(* IEC 61131-3 sources: JaccoSigma/tempclass/Class/DSComm_Interface (part 2) *)

#pragma usingLtd DSComm

#pragma using DSComm

FUNCTION GLOBAL DSComm_Interface::GetVersion
	VAR_OUTPUT
		MessageID 	: DINT;
	END_VAR

  MessageID := DSComm.GetVersion(pThis:=this);
END_FUNCTION

#pragma warning(disable: 73)
FUNCTION VIRTUAL GLOBAL DSComm_Interface::GetVersionResp
	VAR_INPUT
		MessageID 	: DINT;
		ErrorNo 	: DINT;
		pGetVersionRsp 	: ^DSComm::_DS_GetVersionResp;
	END_VAR
#pragma warning(default: 73)

END_FUNCTION

#pragma warning(disable: 73)

#pragma warning(disable: 73)
FUNCTION VIRTUAL GLOBAL DSComm_Interface::GetProjectInfoResp
	VAR_INPUT
		MessageID 	: DINT;
		ErrorNo 	: DINT;
		pGetProjectInfoRsp 	: ^DSComm::_DS_GetProjectInfoResp;
	END_VAR
#pragma warning(default: 73)

END_FUNCTION

FUNCTION GLOBAL DSComm_Interface::UserLogin
	VAR_INPUT
		pUserName 	: ^UINT;
		pPassword 	: ^UINT;
	END_VAR
	VAR_OUTPUT
		MessageID 	: DINT;
	END_VAR

  MessageID := DSComm.UserLogin(pThis:=this, pUserName, pPassword);
END_FUNCTION

#pragma warning(disable: 73)
FUNCTION VIRTUAL GLOBAL DSComm_Interface::UserLoginResp
	VAR_INPUT
    MessageID   : DINT;
    ErrorNo     : DINT;
    pUserLoginData : ^DSComm::_DS_UserLoginResp;
	END_VAR
#pragma warning(default: 73)

END_FUNCTION

FUNCTION GLOBAL DSComm_Interface::GetValue
	VAR_INPUT
		num 	: UDINT;
		pGetValue 	: ^DSComm::_DS_GetValueCmd;
	END_VAR
	VAR_OUTPUT
		MessageID 	: DINT;
	END_VAR

  MessageID := DSComm.GetValue(pThis:=this, num, pGetValue);
END_FUNCTION

#pragma warning(disable: 73)
FUNCTION VIRTUAL GLOBAL DSComm_Interface::GetValueResp
VAR_INPUT
    MessageID   : DINT;
    ErrorNo     : DINT;
    num         : UDINT;
    pGetValueRsp: ^DSComm::_DS_GetValueResp;
END_VAR
#pragma warning(default: 73)

END_FUNCTION

FUNCTION GLOBAL DSComm_Interface::SetValue
	VAR_INPUT
		num 	: UDINT;
		pSetValue 	: ^DSComm::_DS_SetValueCmd;
	END_VAR
	VAR_OUTPUT
		MessageID 	: DINT;
	END_VAR

  MessageID := DSComm.SetValue(pThis:=this, num, pSetValue);
END_FUNCTION

#pragma warning(disable: 73)
FUNCTION VIRTUAL GLOBAL DSComm_Interface::SetValueResp
VAR_INPUT
    MessageID   : DINT;
    ErrorNo     : DINT;
    num         : UDINT;
    pSetValueRsp: ^DSComm::_DS_SetValueResp;
END_VAR
#pragma warning(default: 73)

END_FUNCTION

FUNCTION GLOBAL DSComm_Interface::GetString
	VAR_INPUT
		num 	: UDINT;
		pGetString 	: ^DSComm::_DS_GetStringCmd;
	END_VAR
	VAR_OUTPUT
		MessageID 	: DINT;
	END_VAR

  MessageID := DSComm.GetString(pThis:=this, num, pGetString);
END_FUNCTION

#pragma warning(disable: 73)
FUNCTION VIRTUAL GLOBAL DSComm_Interface::GetStringResp
VAR_INPUT
    MessageID   : DINT;
    ErrorNo     : DINT;
    num         : UDINT;
    pGetStringRsp: ^DSComm::_DS_GetStringResp;
END_VAR
#pragma warning(default: 73)

END_FUNCTION

FUNCTION GLOBAL DSComm_Interface::SetString
	VAR_INPUT
		num 	: UDINT;
		pSetString 	: ^DSComm::_DS_SetStringCmd;
	END_VAR
	VAR_OUTPUT
		MessageID 	: DINT;
	END_VAR

  MessageID := DSComm.SetString(pThis:=this, num, pSetString);
END_FUNCTION

#pragma warning(disable: 73)
FUNCTION VIRTUAL GLOBAL DSComm_Interface::SetStringResp
VAR_INPUT
    MessageID   : DINT;
    ErrorNo     : DINT;
    num         : UDINT;
    pSetStringRsp: ^DSComm::_DS_SetStringResp;
END_VAR
#pragma warning(default: 73)

END_FUNCTION

FUNCTION GLOBAL DSComm_Interface::CancelCommand
	VAR_INPUT
		HandleID 	: DINT;
	END_VAR
	VAR_OUTPUT
		MessageID 	: DINT;
	END_VAR

  MessageID := DSComm.CancelCommand(pThis:=this, HandleID$UDINT);
  MessageID += 1;
END_FUNCTION

#pragma warning(disable: 73)
FUNCTION VIRTUAL GLOBAL DSComm_Interface::CancelCommandResp
	VAR_INPUT
		MessageID 	: DINT;
		ErrorNo 	: DINT;
		pCancelRsp 	: ^DSComm::_DS_CancelResp;
	END_VAR
#pragma warning(default: 73)

END_FUNCTION

FUNCTION GLOBAL DSComm_Interface::Loop
	VAR_INPUT
		Station 	: UDINT;
		pDataSrc 	: pVoid;
		DataLen 	: UDINT;
	END_VAR
	VAR_OUTPUT
		MessageID 	: DINT;
	END_VAR

  MessageID := DSComm.Loop(pThis:=this, Station, pDataSrc, DataLen);
END_FUNCTION

#pragma warning(disable: 73)
FUNCTION VIRTUAL GLOBAL DSComm_Interface::LoopResp
	VAR_INPUT
		MessageID 	: DINT;
		ErrorNo 	: DINT;
		Station 	: UDINT;
		pData 	: pVoid;
		Length 	: UDINT;
	END_VAR
#pragma warning(default: 73)

END_FUNCTION

FUNCTION GLOBAL DSComm_Interface::RecipeLoad
	VAR_INPUT
		pFilterIncl 	: ^DSComm::_DS_UnsLongLongInt;
		pFilterExcl 	: ^DSComm::_DS_UnsLongLongInt;
		crc 	: UDINT;
		pDpne 	: ^CHAR;
	END_VAR
	VAR_OUTPUT
		MessageID 	: DINT;
	END_VAR

  MessageID := DSComm.RecipeLoad(pThis:=this, pFilterIncl, pFilterExcl, crc, pDpne);
END_FUNCTION

#pragma warning(disable: 73)
FUNCTION VIRTUAL GLOBAL DSComm_Interface::RecipeLoadResp
	VAR_INPUT
		MessageID 	: DINT;
		ErrorNo 	: DINT;
		pRecipeLoadRsp 	: ^DSComm::_DS_RecipeLoadResp;
	END_VAR
#pragma warning(default: 73)

END_FUNCTION

FUNCTION GLOBAL DSComm_Interface::RecipeSave
	VAR_INPUT
		pFilterIncl 	: ^DSComm::_DS_UnsLongLongInt;
		pFilterExcl 	: ^DSComm::_DS_UnsLongLongInt;
		pDpne 	: ^CHAR;
		pHeaderText 	: ^CHAR;
	END_VAR
	VAR_OUTPUT
		MessageID 	: DINT;
	END_VAR

  MessageID := DSComm.RecipeSave(pThis:=this, pFilterIncl, pFilterExcl, pDpne, pHeaderText);
END_FUNCTION

#pragma warning(disable: 73)
FUNCTION VIRTUAL GLOBAL DSComm_Interface::RecipeSaveResp
	VAR_INPUT
		MessageID 	: DINT;
		ErrorNo 	: DINT;
		pRecipeSaveRsp 	: ^DSComm::_DS_RecipeSaveResp;
	END_VAR
#pragma warning(default: 73)

END_FUNCTION

FUNCTION GLOBAL DSComm_Interface::SendToAll
	VAR_INPUT
		pDataSrc 	: pVoid;
		DataLen 	: UDINT;
	END_VAR
	VAR_OUTPUT
		MessageID 	: DINT;
	END_VAR

  MessageID := DSComm.SendToAll(pThis:=this, pDataSrc, DataLen);
END_FUNCTION

#pragma warning(disable: 73)
FUNCTION VIRTUAL GLOBAL DSComm_Interface::SendToAllResp
VAR_INPUT
    MessageID   : DINT;
    ErrorNo     : DINT;
END_VAR
#pragma warning(default: 73)

END_FUNCTION

FUNCTION GLOBAL DSComm_Interface::UserLogout
	VAR_OUTPUT
		MessageID 	: DINT;
	END_VAR

  MessageID := DSComm.UserLogout(pThis:=this);
END_FUNCTION

#pragma warning(disable: 73)
FUNCTION VIRTUAL GLOBAL DSComm_Interface::UserLogoutResp
VAR_INPUT
    MessageID   : DINT;
    ErrorNo     : DINT;
END_VAR
#pragma warning(default: 73)

END_FUNCTION

FUNCTION GLOBAL DSComm_Interface::UserPasswordChange
	VAR_INPUT
		pOldPassword 	: ^UINT;
		pNewPassword 	: ^UINT;
	END_VAR
	VAR_OUTPUT
		MessageID 	: DINT;
	END_VAR

  MessageID := DSComm.UserPasswordChange(pThis:=this, pOldPassword, pNewPassword);
END_FUNCTION

#pragma warning(disable: 73)
FUNCTION VIRTUAL GLOBAL DSComm_Interface::UserPasswordChangeResp
	VAR_INPUT
		MessageID 	: DINT;
		ErrorNo 	: DINT;
		pUserPasswordChangeRsp 	: ^DSComm::_DS_UserPasswordChangeResp;
	END_VAR
#pragma warning(default: 73)

END_FUNCTION

FUNCTION GLOBAL DSComm_Interface::CheckAccessLevel
	VAR_INPUT
		num 	: UDINT;
		pCheckAccessLevel 	: ^DSComm::_DS_CheckAccessLevelCmd;
	END_VAR
	VAR_OUTPUT
		MessageID 	: DINT;
	END_VAR

  MessageID := DSComm.CheckAccessLevel(pThis:=this, num, pCheckAccessLevel);
END_FUNCTION

#pragma warning(disable: 73)
FUNCTION VIRTUAL GLOBAL DSComm_Interface::CheckAccessLevelResp
	VAR_INPUT
		MessageID 	: DINT;
		ErrorNo 	: DINT;
		num 	: UDINT;
		pCheckAccessLevelRsp 	: ^DSComm::_DS_CheckAccessLevelResp;
	END_VAR
#pragma warning(default: 73)

END_FUNCTION

FUNCTION GLOBAL DSComm_Interface::CreateUser
	VAR_INPUT
		num 	: UDINT;
		pCreateUser 	: ^DSComm::_DS_CreateUserCmd;
	END_VAR
	VAR_OUTPUT
		MessageID 	: DINT;
	END_VAR

  MessageID := DSComm.CreateUser(pThis:=this, num, pCreateUser);
END_FUNCTION

#pragma warning(disable: 73)
FUNCTION VIRTUAL GLOBAL DSComm_Interface::CreateUserResp
VAR_INPUT
    MessageID   : DINT;
    ErrorNo     : DINT;
    num         : UDINT;
    pCreateUserRsp : ^DSComm::_DS_CreateUserResp;
END_VAR
#pragma warning(default: 73)

END_FUNCTION

FUNCTION GLOBAL DSComm_Interface::ChangeUserSettings
	VAR_INPUT
		num 	: UDINT;
		pChangeUsrSettings 	: ^DSComm::_DS_ChangeUserSettingsCmd;
	END_VAR
	VAR_OUTPUT
		MessageID 	: DINT;
	END_VAR

  MessageID := DSComm.ChangeUserSettings(pThis:=this, num, pChangeUsrSettings);
END_FUNCTION

#pragma warning(disable: 73)
FUNCTION VIRTUAL GLOBAL DSComm_Interface::ChangeUserSettingsResp
	VAR_INPUT
		MessageID 	: DINT;
		ErrorNo 	: DINT;
		num 	: UDINT;
		pChangeUserRsp 	: ^DSComm::_DS_ChangeUserSettingsResp;
	END_VAR
#pragma warning(default: 73)

END_FUNCTION

FUNCTION GLOBAL DSComm_Interface::DeleteUser
	VAR_INPUT
		num 	: UDINT;
		pUserID 	: ^UDINT;
	END_VAR
	VAR_OUTPUT
		MessageID 	: DINT;
	END_VAR

  MessageID := DSComm.DeleteUser(pThis:=this, num, pUserID);
END_FUNCTION

#pragma warning(disable: 73)
FUNCTION VIRTUAL GLOBAL DSComm_Interface::DeleteUserResp
VAR_INPUT
    MessageID   : DINT;
    ErrorNo     : DINT;
    num         : UDINT;
    pDeleteUserRsp : ^DSComm::_DS_DeleteUserResp;
END_VAR
#pragma warning(default: 73)

END_FUNCTION

FUNCTION GLOBAL DSComm_Interface::GetUserList
	VAR_OUTPUT
		MessageID 	: DINT;
	END_VAR

  MessageID := DSComm.GetUserList(pThis:=this);
END_FUNCTION

#pragma warning(disable: 73)
FUNCTION VIRTUAL GLOBAL DSComm_Interface::GetUserListResp
VAR_INPUT
    MessageID   : DINT;
    ErrorNo     : DINT;
    num         : UDINT;
    pGetUserListRsp: ^DSComm::_DS_GetUserListResp;
END_VAR
#pragma warning(default: 73)

END_FUNCTION

FUNCTION GLOBAL DSComm_Interface::GetUserDetails
	VAR_INPUT
		userID 	: UDINT;
	END_VAR
	VAR_OUTPUT
		MessageID 	: DINT;
	END_VAR

  MessageID := DSComm.GetUserDetails(pThis:=this, userID);
END_FUNCTION

#pragma warning(disable: 73)
FUNCTION VIRTUAL GLOBAL DSComm_Interface::GetUserDetailsResp
	VAR_INPUT
		MessageID 	: DINT;
		ErrorNo 	: DINT;
		pUserDetails 	: ^DSComm::_DS_UserLoginResp;
	END_VAR
#pragma warning(default: 73)

END_FUNCTION

FUNCTION GLOBAL DSComm_Interface::CreateRole
	VAR_INPUT
		num 	: UDINT;
		pCreateRolePara 	: ^DSComm::_DS_CreateRoleCmd;
	END_VAR
	VAR_OUTPUT
		MessageID 	: DINT;
	END_VAR

  MessageID := DSComm.CreateRole(pThis:=this, num, pCreateRolePara);
END_FUNCTION

#pragma warning(disable: 73)
FUNCTION VIRTUAL GLOBAL DSComm_Interface::CreateRoleResp
VAR_INPUT
    MessageID   : DINT;
    ErrorNo     : DINT;
    num         : UDINT;
    pCreateRoleRsp : ^DSComm::_DS_CreateRoleResp;
END_VAR
#pragma warning(default: 73)

END_FUNCTION

FUNCTION GLOBAL DSComm_Interface::ChangeRole
	VAR_INPUT
		num 	: UDINT;
		pChangeRole 	: ^DSComm::_DS_ChangeRoleCmd;
	END_VAR
	VAR_OUTPUT
		MessageID 	: DINT;
	END_VAR

  MessageID := DSComm.ChangeRole(pThis:=this, num, pChangeRole);
END_FUNCTION

#pragma warning(disable: 73)
FUNCTION VIRTUAL GLOBAL DSComm_Interface::ChangeRoleResp
VAR_INPUT
    MessageID   : DINT;
    ErrorNo     : DINT;
    num         : UDINT;
    pChangeRoleRsp : ^DSComm::_DS_ChangeRoleResp;
END_VAR
#pragma warning(default: 73)

END_FUNCTION

FUNCTION GLOBAL DSComm_Interface::DeleteRole
	VAR_INPUT
		num 	: UDINT;
		pRoleID 	: ^UDINT;
	END_VAR
	VAR_OUTPUT
		MessageID 	: DINT;
	END_VAR

  MessageID := DSComm.DeleteRole(pThis:=this, num, pRoleID);
END_FUNCTION

#pragma warning(disable: 73)
FUNCTION VIRTUAL GLOBAL DSComm_Interface::DeleteRoleResp
VAR_INPUT
    MessageID   : DINT;
    ErrorNo     : DINT;
    num         : UDINT;
    pDeleteRoleRsp : ^DSComm::_DS_DeleteRoleResp;
END_VAR
#pragma warning(default: 73)

END_FUNCTION

FUNCTION GLOBAL DSComm_Interface::GetRoleList
	VAR_OUTPUT
		MessageID 	: DINT;
	END_VAR

  MessageID := DSComm.GetRoleList(pThis:=this);
END_FUNCTION

#pragma warning(disable: 73)
FUNCTION VIRTUAL GLOBAL DSComm_Interface::GetRoleListResp
VAR_INPUT
    MessageID   : DINT;
    ErrorNo     : DINT;
    num         : UDINT;
    pGetRoleListRsp: ^DSComm::_DS_GetRoleListResp;
END_VAR
#pragma warning(default: 73)

END_FUNCTION

FUNCTION GLOBAL DSComm_Interface::GetRoleDetails
	VAR_INPUT
		roleID 	: UDINT;
	END_VAR
	VAR_OUTPUT
		MessageID 	: DINT;
	END_VAR

  MessageID := DSComm.GetRoleDetails(pThis:=this, roleID);
END_FUNCTION

#pragma warning(disable: 73)
FUNCTION VIRTUAL GLOBAL DSComm_Interface::GetRoleDetailsResp
VAR_INPUT
    MessageID   : DINT;
    ErrorNo     : DINT;
    pGetRoleDetailsRsp : ^DSComm::_DS_GetRoleDetailsResp;
END_VAR
#pragma warning(default: 73)

END_FUNCTION

FUNCTION GLOBAL DSComm_Interface::GetVarIdFromName
	VAR_INPUT
		num 	: UDINT;
		ppName 	: ^pChar;
	END_VAR
	VAR_OUTPUT
		MessageID 	: DINT;
	END_VAR

  MessageID := DSComm.GetVarIdFromName(pThis:=this, num, ppName);
END_FUNCTION

#pragma warning(disable: 73)
FUNCTION VIRTUAL GLOBAL DSComm_Interface::GetVarIdFromNameResp
VAR_INPUT
    MessageID   : DINT;
    ErrorNo     : DINT;
    num         : UDINT;
    pGetVarIdFromNameRsp: ^DSComm::_DS_GetVarIdFromNameResp;
END_VAR
#pragma warning(default: 73)

END_FUNCTION

FUNCTION GLOBAL DSComm_Interface::GetVarIdFromLasalId
	VAR_INPUT
		num 	: UDINT;
		pLasalId 	: ^DSComm::_DS_GetVarIdFromLasalIdCmd;
	END_VAR
	VAR_OUTPUT
		MessageID 	: DINT;
	END_VAR

  MessageID := DSComm.GetVarIdFromLasalId(pThis:=this, num, pLasalId);
END_FUNCTION

#pragma warning(disable: 73)
FUNCTION VIRTUAL GLOBAL DSComm_Interface::GetVarIdFromLasalIdResp
VAR_INPUT
    MessageID   : DINT;
    ErrorNo     : DINT;
    num         : UDINT;
    pGetVarIdFromLasalIdRsp: ^DSComm::_DS_GetVarIdFromLasalIdResp;
END_VAR
#pragma warning(default: 73)

END_FUNCTION

FUNCTION GLOBAL DSComm_Interface::GetLasalIdFromName
	VAR_INPUT
		num 	: UDINT;
		ppName 	: ^pChar;
	END_VAR
	VAR_OUTPUT
		MessageID 	: DINT;
	END_VAR

  MessageID := DSComm.GetLasalIdFromName(pThis:=this, num, ppName);
END_FUNCTION

#pragma warning(disable: 73)
FUNCTION VIRTUAL GLOBAL DSComm_Interface::GetLasalIdFromNameResp
VAR_INPUT
    MessageID   : DINT;
    ErrorNo     : DINT;
    num         : UDINT;
    pGetLasalIdFromNameRsp: ^DSComm::_DS_GetLasalIdFromNameResp;
END_VAR
#pragma warning(default: 73)

END_FUNCTION

FUNCTION GLOBAL DSComm_Interface::GetLasalIdFromVarId
	VAR_INPUT
		num 	: UDINT;
		pVarId 	: ^UDINT;
	END_VAR
	VAR_OUTPUT
		MessageID 	: DINT;
	END_VAR

  MessageID := DSComm.GetLasalIdFromVarId(pThis:=this, num, pVarId);
END_FUNCTION

#pragma warning(disable: 73)
FUNCTION VIRTUAL GLOBAL DSComm_Interface::GetLasalIdFromVarIdResp
VAR_INPUT
    MessageID   : DINT;
    ErrorNo     : DINT;
    num         : UDINT;
    pGetLasalIdIdFromVarIdRsp: ^DSComm::_DS_GetLasalIdIdFromVarIdResp;
END_VAR
#pragma warning(default: 73)

END_FUNCTION

FUNCTION GLOBAL DSComm_Interface::GetNameFromVarId
	VAR_INPUT
		num 	: UDINT;
		pVarId 	: ^UDINT;
	END_VAR
	VAR_OUTPUT
		MessageID 	: DINT;
	END_VAR

  MessageID := DSComm.GetNameFromVarId(pThis:=this, num, pVarId);
END_FUNCTION

#pragma warning(disable: 73)
FUNCTION VIRTUAL GLOBAL DSComm_Interface::GetNameFromVarIdResp
VAR_INPUT
    MessageID   : DINT;
    ErrorNo     : DINT;
    num         : UDINT;
    pGetNameFromVarIdRsp: ^DSComm::_DS_GetNameFromVarIdResp;
END_VAR
#pragma warning(default: 73)

END_FUNCTION

FUNCTION GLOBAL DSComm_Interface::GetNameFromLasalId
	VAR_INPUT
		num 	: UDINT;
		pLasalId 	: ^DSComm::_DS_GetNameFromLasalIdCmd;
	END_VAR
	VAR_OUTPUT
		MessageID 	: DINT;
	END_VAR

  MessageID := DSComm.GetNameFromLasalId(pThis:=this, num, pLasalId);
END_FUNCTION

#pragma warning(disable: 73)
FUNCTION VIRTUAL GLOBAL DSComm_Interface::GetNameFromLasalIdResp
VAR_INPUT
    MessageID   : DINT;
    ErrorNo     : DINT;
    num         : UDINT;
    pGetNameFromLasalIdRsp: ^DSComm::_DS_GetNameFromLasalIdResp;
END_VAR
#pragma warning(default: 73)

END_FUNCTION

FUNCTION GLOBAL DSComm_Interface::IncValue
	VAR_INPUT
		num 	: UDINT;
		pdpId : ^UDINT;
	END_VAR
	VAR_OUTPUT
		MessageID 	: DINT;
	END_VAR

  MessageID := DSComm.IncValue(pThis:=this, num, pdpId);
END_FUNCTION

#pragma warning(disable: 73)
FUNCTION VIRTUAL GLOBAL DSComm_Interface::IncValueResp
VAR_INPUT
    MessageID   : DINT;
    ErrorNo     : DINT;
    num         : UDINT;
    pIncValueRsp: ^DSComm::_DS_IncDecValueResp;
END_VAR
#pragma warning(default: 73)

END_FUNCTION

FUNCTION GLOBAL DSComm_Interface::DecValue
	VAR_INPUT
		num 	: UDINT;
		pdpId : ^UDINT;
	END_VAR
	VAR_OUTPUT
		MessageID 	: DINT;
	END_VAR

  MessageID := DSComm.DecValue(pThis:=this, num, pdpId);
END_FUNCTION

#pragma warning(disable: 73)
FUNCTION VIRTUAL GLOBAL DSComm_Interface::DecValueResp
VAR_INPUT
    MessageID   : DINT;
    ErrorNo     : DINT;
    num         : UDINT;
    pDecValueRsp: ^DSComm::_DS_IncDecValueResp;
END_VAR
#pragma warning(default: 73)

END_FUNCTION

FUNCTION GLOBAL DSComm_Interface::RefListAdd
	VAR_INPUT
		channel 	: UDINT;
		num 	: UDINT;
		pDpId 	: ^UDINT;
	END_VAR
	VAR_OUTPUT
		MessageID 	: DINT;
	END_VAR

  MessageID := DSComm.RefListAdd(pThis:=this, channel, num, pDpId);
END_FUNCTION

#pragma warning(disable: 73)
FUNCTION VIRTUAL GLOBAL DSComm_Interface::RefListAddResp
	VAR_INPUT
		MessageID 	: DINT;
		ErrorNo 	: DINT;
		Channel 	: UDINT;
		num 	: UDINT;
		pRefListAddRsp 	: ^DSComm::_DS_RefListAddResp;
	END_VAR
#pragma warning(default: 73)

END_FUNCTION

FUNCTION GLOBAL DSComm_Interface::RefListSub
	VAR_INPUT
		channel 	: UDINT;
		num 	: UDINT;
		pDpId 	: ^UDINT;
	END_VAR
	VAR_OUTPUT
		MessageID 	: DINT;
	END_VAR

  MessageID := DSComm.RefListSub(pThis:=this, channel, num, pDpId);
END_FUNCTION

#pragma warning(disable: 73)
FUNCTION VIRTUAL GLOBAL DSComm_Interface::RefListSubResp
	VAR_INPUT
		MessageID 	: DINT;
		ErrorNo 	: DINT;
		Channel 	: UDINT;
		num 	: UDINT;
		pRefListSubRsp 	: ^DSComm::_DS_RefListSubResp;
	END_VAR
#pragma warning(default: 73)

END_FUNCTION

#pragma warning(disable: 73)
FUNCTION VIRTUAL GLOBAL DSComm_Interface::RefListUpdatePush
	VAR_INPUT
		ErrorNo 	: DINT;
		channel 	: UDINT;
		num 	: UDINT;
		pRefListUpdate 	: ^DSComm::_DS_RefListUpdate;
	END_VAR
#pragma warning(default: 73)

END_FUNCTION

#pragma warning(disable: 73)
FUNCTION VIRTUAL GLOBAL DSComm_Interface::RefListUpdateStringPush
	VAR_INPUT
		ErrorNo 	: DINT;
		channel 	: UDINT;
		num 	: UDINT;
		pRefListUpdateString 	: ^DSComm::_DS_RefListUpdateString;
	END_VAR
#pragma warning(default: 73)

END_FUNCTION

FUNCTION GLOBAL DSComm_Interface::GetDpInfo
	VAR_INPUT
		num 	: UDINT;
		pVarId 	: ^UDINT;
	END_VAR
	VAR_OUTPUT
		MessageID 	: DINT;
	END_VAR

  MessageID := DSComm.GetDpInfo(pThis:=this, num, pVarId);
END_FUNCTION

#pragma warning(disable: 73)
FUNCTION VIRTUAL GLOBAL DSComm_Interface::GetDpInfoResp
VAR_INPUT
    MessageID   : DINT;
    ErrorNo     : DINT;
    num         : UDINT;
    pGetDpInfoRsp: ^DSComm::_DS_GetDpInfoResp;
END_VAR
#pragma warning(default: 73)

END_FUNCTION

FUNCTION GLOBAL DSComm_Interface::GetDpList
	VAR_INPUT
		pFilterIncl 	: ^DSComm::_DS_UnsLongLongInt;
		pFilterExcl 	: ^DSComm::_DS_UnsLongLongInt;
	END_VAR
	VAR_OUTPUT
		MessageID 	: DINT;
	END_VAR

  MessageID := DSComm.GetDpList(pThis:=this, pFilterIncl, pFilterExcl);
END_FUNCTION

#pragma warning(disable: 73)
FUNCTION VIRTUAL GLOBAL DSComm_Interface::GetDpListResp
	VAR_INPUT
		MessageID 	: DINT;
		ErrorNo 	: DINT;
		TotalNum 	: UDINT;
		num 	: UDINT;
		LastPacket 	: BOOL;
		pGetDpListRsp 	: ^DSComm::_DS_GetDpListResp;
	END_VAR
#pragma warning(default: 73)

END_FUNCTION

#pragma warning(disable: 73)

#pragma warning(disable: 73)

FUNCTION GLOBAL DSComm_Interface::FileOpen
	VAR_INPUT
		pDpne 	: ^CHAR;
		pMode 	: ^CHAR;
	END_VAR
	VAR_OUTPUT
		MessageID 	: DINT;
	END_VAR

  MessageID := DSComm.FileOpen(pThis:=this, pDpne, pMode);
END_FUNCTION

#pragma warning(disable: 73)
FUNCTION VIRTUAL GLOBAL DSComm_Interface::FileOpenResp
VAR_INPUT
    MessageID   : DINT;
    ErrorNo     : DINT;
    pFileOpenRsp: ^DSComm::_DS_FileOpenResp;
END_VAR
#pragma warning(default: 73)

END_FUNCTION

FUNCTION GLOBAL DSComm_Interface::FileClose
	VAR_INPUT
		handle 	: UDINT;
	END_VAR
	VAR_OUTPUT
		MessageID 	: DINT;
	END_VAR

  MessageID := DSComm.FileClose(pThis:=this, handle);
END_FUNCTION

#pragma warning(disable: 73)
FUNCTION VIRTUAL GLOBAL DSComm_Interface::FileCloseResp
VAR_INPUT
    MessageID   : DINT;
    ErrorNo     : DINT;
    pFileCloseRsp: ^DSComm::_DS_FileCloseResp;
END_VAR
#pragma warning(default: 73)

END_FUNCTION

FUNCTION GLOBAL DSComm_Interface::FileSeek
	VAR_INPUT
		handle 	: UDINT;
		start 	: UDINT;
		offset 	: UDINT;
	END_VAR
	VAR_OUTPUT
		MessageID 	: DINT;
	END_VAR

  MessageID := DSComm.FileSeek(pThis:=this, handle, start, offset);
END_FUNCTION

#pragma warning(disable: 73)
FUNCTION VIRTUAL GLOBAL DSComm_Interface::FileSeekResp
VAR_INPUT
    MessageID   : DINT;
    ErrorNo     : DINT;
    pFileSeekRsp: ^DSComm::_DS_FileSeekResp;
END_VAR
#pragma warning(default: 73)

END_FUNCTION

FUNCTION GLOBAL DSComm_Interface::FileTell
	VAR_INPUT
		handle 	: UDINT;
	END_VAR
	VAR_OUTPUT
		MessageID 	: DINT;
	END_VAR

  MessageID := DSComm.FileTell(pThis:=this, handle);
END_FUNCTION

#pragma warning(disable: 73)
FUNCTION VIRTUAL GLOBAL DSComm_Interface::FileTellResp
	VAR_INPUT
		MessageID 	: DINT;
		ErrorNo 	: DINT;
		pFileTellRsp 	: ^DSComm::_DS_FileTellResp;
	END_VAR
#pragma warning(default: 73)

END_FUNCTION

FUNCTION GLOBAL DSComm_Interface::FileRead
	VAR_INPUT
		handle 	: UDINT;
		length 	: UDINT;
	END_VAR
	VAR_OUTPUT
		MessageID 	: DINT;
	END_VAR

  MessageID := DSComm.FileRead(pThis:=this, handle, length);
END_FUNCTION

#pragma warning(disable: 73)
FUNCTION VIRTUAL GLOBAL DSComm_Interface::FileReadResp
VAR_INPUT
    MessageID   : DINT;
    ErrorNo     : DINT;
    pFileReadRsp: ^DSComm::_DS_FileReadResp;
END_VAR
#pragma warning(default: 73)

END_FUNCTION

FUNCTION GLOBAL DSComm_Interface::FileWrite
	VAR_INPUT
		handle 	: UDINT;
		length 	: UDINT;
		pWriteData 	: ^CHAR;
	END_VAR
	VAR_OUTPUT
		MessageID 	: DINT;
	END_VAR

  MessageID := DSComm.FileWrite(pThis:=this, handle, length, pWriteData);
END_FUNCTION

#pragma warning(disable: 73)
FUNCTION VIRTUAL GLOBAL DSComm_Interface::FileWriteResp
VAR_INPUT
    MessageID   : DINT;
    ErrorNo     : DINT;
    pFileWriteRsp: ^DSComm::_DS_FileWriteResp;
END_VAR
#pragma warning(default: 73)

END_FUNCTION

FUNCTION GLOBAL DSComm_Interface::FileGet
	VAR_INPUT
		handle 	: UDINT;
		length 	: UDINT;
	END_VAR
	VAR_OUTPUT
		MessageID 	: DINT;
	END_VAR

  MessageID := DSComm.FileGet(pThis:=this, handle, length);
END_FUNCTION

#pragma warning(disable: 73)
FUNCTION VIRTUAL GLOBAL DSComm_Interface::FileGetResp
VAR_INPUT
    MessageID   : DINT;
    ErrorNo     : DINT;
    pFileGetRsp: ^DSComm::_DS_FileGetResp;
END_VAR
#pragma warning(default: 73)

END_FUNCTION

FUNCTION GLOBAL DSComm_Interface::FilePut
	VAR_INPUT
		handle 	: UDINT;
		pString 	: ^CHAR;
	END_VAR
	VAR_OUTPUT
		MessageID 	: DINT;
	END_VAR

  MessageID := DSComm.FilePut(pThis:=this, handle, pString);
END_FUNCTION

#pragma warning(disable: 73)
FUNCTION VIRTUAL GLOBAL DSComm_Interface::FilePutResp
VAR_INPUT
    MessageID   : DINT;
    ErrorNo     : DINT;
    pFilePutRsp: ^DSComm::_DS_FilePutResp;
END_VAR
#pragma warning(default: 73)

END_FUNCTION

FUNCTION GLOBAL DSComm_Interface::FileLength
	VAR_INPUT
		handle 	: UDINT;
	END_VAR
	VAR_OUTPUT
		MessageID 	: DINT;
	END_VAR

  MessageID := DSComm.FileLength(pThis:=this, handle);
END_FUNCTION

#pragma warning(disable: 73)
FUNCTION VIRTUAL GLOBAL DSComm_Interface::FileLengthResp
	VAR_INPUT
		MessageID 	: DINT;
		ErrorNo 	: DINT;
		pFileLengthRsp 	: ^DSComm::_DS_FileLengthResp;
	END_VAR
#pragma warning(default: 73)

END_FUNCTION

FUNCTION GLOBAL DSComm_Interface::FileContent
	VAR_INPUT
		pDpne 	: ^CHAR;
	END_VAR
	VAR_OUTPUT
		MessageID 	: DINT;
	END_VAR

  MessageID := DSComm.FileContent(pThis:=this, pDpne);
END_FUNCTION

#pragma warning(disable: 73)
FUNCTION VIRTUAL GLOBAL DSComm_Interface::FileContentResp
	VAR_INPUT
		MessageID 	: DINT;
		ErrorNo 	: DINT;
		LastPacket 	: BOOL;
		pFileContentRsp 	: ^DSComm::_DS_FileContentResp;
	END_VAR
#pragma warning(default: 73)

END_FUNCTION

FUNCTION GLOBAL DSComm_Interface::DirCreate
	VAR_INPUT
		pDp 	: ^CHAR;
	END_VAR
	VAR_OUTPUT
		MessageID 	: DINT;
	END_VAR

  MessageID := DSComm.DirCreate(pThis:=this, pDp);
END_FUNCTION

#pragma warning(disable: 73)
FUNCTION VIRTUAL GLOBAL DSComm_Interface::DirCreateResp
VAR_INPUT
    MessageID   : DINT;
    ErrorNo     : DINT;
    pDirCreateRsp: ^DSComm::_DS_DirCreateResp;
END_VAR
#pragma warning(default: 73)

END_FUNCTION

FUNCTION GLOBAL DSComm_Interface::DirRead
	VAR_INPUT
		FilterIncl 	: UDINT;
		FilterExcl 	: UDINT;
		pDp 	: ^CHAR;
		pNe 	: ^CHAR;
	END_VAR
	VAR_OUTPUT
		MessageID 	: DINT;
	END_VAR

  MessageID := DSComm.DirRead(pThis:=this, FilterIncl, FilterExcl, pDp, pNe);
END_FUNCTION

#pragma warning(disable: 73)
FUNCTION VIRTUAL GLOBAL DSComm_Interface::DirReadResp
	VAR_INPUT
		MessageID 	: DINT;
		ErrorNo 	: DINT;
		DS_ErrorNo 	: DINT;
		num 	: UDINT;
		LastPacket 	: BOOL;
		pDirReadRsp 	: ^DSComm::_DS_DirReadResp;
	END_VAR
#pragma warning(default: 73)

END_FUNCTION

FUNCTION GLOBAL DSComm_Interface::FileRemove
	VAR_INPUT
		pDpne 	: ^CHAR;
		updateProgress 	: BOOL;
	END_VAR
	VAR_OUTPUT
		MessageID 	: DINT;
	END_VAR

  MessageID := DSComm.FileRemove(pThis:=this, pDpne, updateProgress);
END_FUNCTION

#pragma warning(disable: 73)
FUNCTION VIRTUAL GLOBAL DSComm_Interface::FileRemoveResp
VAR_INPUT
    MessageID   : DINT;
    ErrorNo     : DINT;
    pFileRemoveRsp: ^DSComm::_DS_FileRemoveResp;
END_VAR
#pragma warning(default: 73)

END_FUNCTION

FUNCTION GLOBAL DSComm_Interface::FileCopy
	VAR_INPUT
		pDpneSrc 	: ^CHAR;
		pDpneDest 	: ^CHAR;
		updateProgress 	: BOOL;
	END_VAR
	VAR_OUTPUT
		MessageID 	: DINT;
	END_VAR

  MessageID := DSComm.FileCopy(pThis:=this, pDpneSrc, pDpneDest, updateProgress);
END_FUNCTION

#pragma warning(disable: 73)
FUNCTION VIRTUAL GLOBAL DSComm_Interface::FileCopyResp
VAR_INPUT
    MessageID   : DINT;
    ErrorNo     : DINT;
    pFileCopyRsp: ^DSComm::_DS_FileCopyResp;
END_VAR
#pragma warning(default: 73)

END_FUNCTION

FUNCTION GLOBAL DSComm_Interface::FileInfo
	VAR_INPUT
		pDpne 	: ^CHAR;
	END_VAR
	VAR_OUTPUT
		MessageID 	: DINT;
	END_VAR

  MessageID := DSComm.FileInfo(pThis:=this, pDpne);
END_FUNCTION

#pragma warning(disable: 73)
FUNCTION VIRTUAL GLOBAL DSComm_Interface::FileInfoResp
VAR_INPUT
    MessageID   : DINT;
    ErrorNo     : DINT;
    pFileInfoRsp: ^DSComm::_DS_FileInfoResp;
END_VAR
#pragma warning(default: 73)

END_FUNCTION

FUNCTION GLOBAL DSComm_Interface::FileRename
	VAR_INPUT
		pDpneOld 	: ^CHAR;
		pDpneNew 	: ^CHAR;
	END_VAR
	VAR_OUTPUT
		MessageID 	: DINT;
	END_VAR

  MessageID := DSComm.FileRename(pThis:=this, pDpneOld, pDpneNew);
END_FUNCTION

#pragma warning(disable: 73)
FUNCTION VIRTUAL GLOBAL DSComm_Interface::FileRenameResp
VAR_INPUT
    MessageID   : DINT;
    ErrorNo     : DINT;
    pFileRenameRsp: ^DSComm::_DS_FileRenameResp;
END_VAR
#pragma warning(default: 73)

END_FUNCTION

FUNCTION GLOBAL DSComm_Interface::FileSetAttribute
	VAR_INPUT
		pDpne 	: ^CHAR;
		AttributeToSet 	: UDINT;
		AttributeToReset 	: UDINT;
	END_VAR
	VAR_OUTPUT
		MessageID 	: DINT;
	END_VAR

  MessageID := DSComm.FileSetAttribute(pThis:=this, pDpne, AttributeToSet, AttributeToReset);
END_FUNCTION

#pragma warning(disable: 73)
FUNCTION VIRTUAL GLOBAL DSComm_Interface::FileSetAttributeResp
VAR_INPUT
    MessageID   : DINT;
    ErrorNo     : DINT;
    pFileSetAttributeRsp: ^DSComm::_DS_FileSetAttributeResp;
END_VAR
#pragma warning(default: 73)

END_FUNCTION

FUNCTION GLOBAL DSComm_Interface::GetDriveList
	VAR_OUTPUT
		MessageID 	: DINT;
	END_VAR

  MessageID := DSComm.GetDriveList(pThis:=this);
END_FUNCTION

#pragma warning(disable: 73)
FUNCTION VIRTUAL GLOBAL DSComm_Interface::GetDriveListResp
VAR_INPUT
    MessageID   : DINT;
    ErrorNo     : DINT;
    pGetDriveListRsp: ^DSComm::_DS_GetDriveListResp;
END_VAR
#pragma warning(default: 73)

END_FUNCTION

FUNCTION GLOBAL DSComm_Interface::FileMove
	VAR_INPUT
		pDpneSrc 	: ^CHAR;
		pDpneDest 	: ^CHAR;
		updateProgress 	: BOOL;
	END_VAR
	VAR_OUTPUT
		MessageID 	: DINT;
	END_VAR

  MessageID := DSComm.FileMove(pThis:=this, pDpneSrc, pDpneDest, updateProgress);
END_FUNCTION

#pragma warning(disable: 73)
FUNCTION VIRTUAL GLOBAL DSComm_Interface::FileMoveResp
VAR_INPUT
    MessageID   : DINT;
    ErrorNo     : DINT;
    pFileMoveRsp:^DSComm::_DS_FileMoveResp;
END_VAR
#pragma warning(default: 73)

END_FUNCTION

FUNCTION GLOBAL DSComm_Interface::EventjournalAdd
	VAR_INPUT
		num 	: UDINT;
		pEventjournalAdd 	: ^DSComm::_DS_EventjournalAddCmd;
	END_VAR
	VAR_OUTPUT
		MessageID 	: DINT;
	END_VAR

  MessageID := DSComm.EventjournalAdd(pThis:=this, num, pEventjournalAdd);
END_FUNCTION

#pragma warning(disable: 73)
FUNCTION VIRTUAL GLOBAL DSComm_Interface::EventjournalAddResp
VAR_INPUT
    MessageID   : DINT;
    ErrorNo     : DINT;
    num         : UDINT;
    pEventjournalAddRsp: ^DSComm::_DS_EventjournalAddResp;
END_VAR
#pragma warning(default: 73)

END_FUNCTION

FUNCTION GLOBAL DSComm_Interface::EventjournalGet
	VAR_INPUT
		num 	: UDINT;
		pJournalId 	: ^UDINT;
	END_VAR
	VAR_OUTPUT
		MessageID 	: DINT;
	END_VAR

  MessageID := DSComm.EventjournalGet(pThis:=this, num, pJournalId);
END_FUNCTION

#pragma warning(disable: 73)
FUNCTION VIRTUAL GLOBAL DSComm_Interface::EventjournalGetResp
VAR_INPUT
    MessageID   : DINT;
    ErrorNo     : DINT;
    num         : UDINT;
    pEventjournalGetRsp: ^DSComm::_DS_EventjournalGetResp;
END_VAR
#pragma warning(default: 73)

END_FUNCTION

FUNCTION GLOBAL DSComm_Interface::EventjournalGetAll
	VAR_OUTPUT
		MessageID 	: DINT;
	END_VAR

  MessageID := DSComm.EventjournalGetAll(pThis:=this);
END_FUNCTION

#pragma warning(disable: 73)
FUNCTION VIRTUAL GLOBAL DSComm_Interface::EventjournalGetAllResp
	VAR_INPUT
		MessageID 	: DINT;
		ErrorNo 	: DINT;
		num 	: UDINT;
		LastPacket 	: BOOL;
		pEventjournalGetAllRsp 	: ^DSComm::_DS_EventjournalGetResp;
	END_VAR
#pragma warning(default: 73)

END_FUNCTION

FUNCTION GLOBAL DSComm_Interface::EventjournalDel
	VAR_INPUT
		num 	: UDINT;
		pJournalId 	: ^UDINT;
	END_VAR
	VAR_OUTPUT
		MessageID 	: DINT;
	END_VAR

  MessageID := DSComm.EventjournalDel(pThis:=this, num, pJournalId);
END_FUNCTION

#pragma warning(disable: 73)
FUNCTION VIRTUAL GLOBAL DSComm_Interface::EventjournalDelResp
VAR_INPUT
    MessageID   : DINT;
    ErrorNo     : DINT;
    num         : UDINT;
    pEventjournalDelRsp: ^DSComm::_DS_EventjournalDelResp;
END_VAR
#pragma warning(default: 73)

END_FUNCTION

FUNCTION GLOBAL DSComm_Interface::EventjournalDelAll
	VAR_OUTPUT
		MessageID 	: DINT;
	END_VAR

  MessageID := DSComm.EventjournalDelAll(pThis:=this);
END_FUNCTION

#pragma warning(disable: 73)
FUNCTION VIRTUAL GLOBAL DSComm_Interface::EventjournalDelAllResp
	VAR_INPUT
		MessageID 	: DINT;
		ErrorNo 	: DINT;
		num 	: UDINT;
		pEventjournalDelAllRsp 	: ^DSComm::_DS_EventjournalDelAllResp;
	END_VAR
#pragma warning(default: 73)

END_FUNCTION

#pragma warning(disable: 73)
FUNCTION VIRTUAL GLOBAL DSComm_Interface::EventjournalUpdatePush
	VAR_INPUT
		MessageID 	: DINT;
		ErrorNo 	: DINT;
		num 	: UDINT;
		pEventjournalUpd 	: ^DSComm::_DS_EventjournalGetResp;
	END_VAR
#pragma warning(default: 73)

END_FUNCTION

FUNCTION GLOBAL DSComm_Interface::EventjournalQuitAlarm
	VAR_INPUT
		num 	: UDINT;
		pAlarmId 	: ^UDINT;
	END_VAR
	VAR_OUTPUT
		MessageID 	: DINT;
	END_VAR

  MessageID := DSComm.EventjournalQuitAlarm(pThis:=this, num, pAlarmId);
END_FUNCTION

#pragma warning(disable: 73)
FUNCTION VIRTUAL GLOBAL DSComm_Interface::EventjournalQuitAlarmResp
VAR_INPUT
    MessageID   : DINT;
    ErrorNo     : DINT;
    num         : UDINT;
    pEventjournalQuitAlarmRsp: ^DSComm::_DS_EventjournalQuitAlarmResp;
END_VAR
#pragma warning(default: 73)

END_FUNCTION

FUNCTION GLOBAL DSComm_Interface::EventjournalQuitAll
	VAR_OUTPUT
		MessageID 	: DINT;
	END_VAR

  MessageID := DSComm.EventjournalQuitAll(pThis:=this);
END_FUNCTION

#pragma warning(disable: 73)
FUNCTION VIRTUAL GLOBAL DSComm_Interface::EventjournalQuitAllResp
VAR_INPUT
    MessageID   : DINT;
    ErrorNo     : DINT;
    num         : UDINT;
    pEventjournalQuitAllRsp: ^DSComm::_DS_EventjournalQuitAllResp;
END_VAR
#pragma warning(default: 73)

END_FUNCTION

FUNCTION GLOBAL DSComm_Interface::ResetDataservice
	VAR_OUTPUT
		MessageID 	: DINT;
	END_VAR

  MessageID := DSComm.ResetDataservice(pThis:=this);
END_FUNCTION

#pragma warning(disable: 73)
FUNCTION VIRTUAL GLOBAL DSComm_Interface::ResetDataserviceResp
VAR_INPUT
    MessageID   : DINT;
    ErrorNo     : DINT;
    pResetDataserviceRsp : ^DSComm::_DS_ResetDataserviceResp;
END_VAR
#pragma warning(default: 73)

END_FUNCTION

FUNCTION GLOBAL DSComm_Interface::RestartDataservice
	VAR_OUTPUT
		MessageID 	: DINT;
	END_VAR

  MessageID := DSComm.RestartDataservice(pThis:=this);
END_FUNCTION

#pragma warning(disable: 73)
FUNCTION VIRTUAL GLOBAL DSComm_Interface::RestartDataserviceResp
VAR_INPUT
    MessageID   : DINT;
    ErrorNo     : DINT;
    pRestartDataserviceRsp : ^DSComm::_DS_RestartDataserviceResp;
END_VAR
#pragma warning(default: 73)

END_FUNCTION

FUNCTION GLOBAL DSComm_Interface::GetStationStatus
	VAR_INPUT
		num 	: UDINT;
		pStationNo 	: ^UDINT;
	END_VAR
	VAR_OUTPUT
		MessageID 	: DINT;
	END_VAR

  MessageID := DSComm.GetStationStatus(pThis:=this, num, pStationNo);
END_FUNCTION

#pragma warning(disable: 73)
FUNCTION VIRTUAL GLOBAL DSComm_Interface::GetStationStatusResp
VAR_INPUT
    MessageID   : DINT;
    ErrorNo     : DINT;
    num         : UDINT;
    pStationStatusRsp: ^DSComm::_DS_StationStatusResp;
END_VAR
#pragma warning(default: 73)

END_FUNCTION

FUNCTION GLOBAL DSComm_Interface::GetVarIdFromCRC
	VAR_INPUT
		num 	: UDINT;
		pCRC 	: ^UDINT;
	END_VAR
	VAR_OUTPUT
		MessageID 	: DINT;
	END_VAR

  MessageID := DSComm.GetVarIdFromCRC(pThis:=this, num, pCRC);
END_FUNCTION

#pragma warning(disable: 73)
FUNCTION VIRTUAL GLOBAL DSComm_Interface::GetVarIdFromCRCResp
VAR_INPUT
    MessageID   : DINT;
    ErrorNo     : DINT;
    num         : UDINT;
    pGetVarIdFromCRCRsp: ^DSComm::_DS_GetVarIdFromCRCResp;
END_VAR
#pragma warning(default: 73)

END_FUNCTION

FUNCTION GLOBAL DSComm_Interface::GetCRCfromVarId
	VAR_INPUT
		num 	: UDINT;
		pVarId 	: ^UDINT;
	END_VAR
	VAR_OUTPUT
		MessageID 	: DINT;
	END_VAR

  MessageID := DSComm.GetCRCfromVarId(pThis:=this, num, pVarId);
END_FUNCTION

#pragma warning(disable: 73)
FUNCTION VIRTUAL GLOBAL DSComm_Interface::GetCRCfromVarIdResp
VAR_INPUT
    MessageID   : DINT;
    ErrorNo     : DINT;
    num         : UDINT;
    pGetCRCfromVarIdRsp: ^DSComm::_DS_GetCRCfromVarIdResp;
END_VAR
#pragma warning(default: 73)

END_FUNCTION

FUNCTION GLOBAL DSComm_Interface::IsConnected
	VAR_OUTPUT
		OutParam 	: BOOL;
	END_VAR

  OutParam := DSComm.IsConnected();
END_FUNCTION

FUNCTION GLOBAL DSComm_Interface::GetLoginInfo
	VAR_OUTPUT
		userID 	: UDINT;
	END_VAR

  userID := DSComm.GetLoginInfo();
END_FUNCTION

#pragma warning(disable: 73)
FUNCTION VIRTUAL GLOBAL DSComm_Interface::ProgressStatusPush
	VAR_INPUT
		pProgressStatus 	: ^DSComm::_DS_ProgressStatus;
	END_VAR
#pragma warning(default: 73)

END_FUNCTION

#pragma warning(disable: 73)
FUNCTION VIRTUAL GLOBAL DSComm_Interface::GetStationListResp
	VAR_INPUT
		MessageID 	: DINT;
		ErrorNo 	: DINT;
		num 	: UDINT;
		pGetStationListRsp 	: ^DSComm::_DS_StationListResp;
	END_VAR
#pragma warning(default: 73)

END_FUNCTION

FUNCTION GLOBAL DSComm_Interface::GetStationList
	VAR_OUTPUT
		MessageID 	: DINT;
	END_VAR

  MessageID := DSComm.GetStationList(pThis:=this);
END_FUNCTION

#pragma warning(disable: 73)
FUNCTION VIRTUAL GLOBAL DSComm_Interface::SendToAllPush
	VAR_INPUT
		MessageID 	: DINT;
		ErrorNo 	: DINT;
		pData 	: ^CHAR;
		Length 	: UDINT;
	END_VAR
#pragma warning(default: 73)

END_FUNCTION

FUNCTION GLOBAL DSComm_Interface::SendUserEvent
	VAR_INPUT
		MajorID 	: UINT;
		MinorID 	: UINT;
		SessionID 	: UINT;
		pDataSrc 	: pVoid;
		DataLen 	: UDINT;
	END_VAR
	VAR_OUTPUT
		MessageID 	: DINT;
	END_VAR

  MessageID := DSComm.SendUserEvent(pThis:=this, MajorID, MinorID, SessionID, pDataSrc, DataLen);
END_FUNCTION

#pragma warning(disable: 73)
FUNCTION VIRTUAL GLOBAL DSComm_Interface::SendUserEventResp
	VAR_INPUT
		MessageID 	: DINT;
		ErrorNo 	: DINT;
		pUserEventRsp 	: ^DSComm::_DS_UserEventResp;
	END_VAR
#pragma warning(default: 73)

END_FUNCTION

FUNCTION GLOBAL DSComm_Interface::SubscribeEventjournalUpdates

  DSComm.SubscribeEventjournalUpdates(pThis:=this);

END_FUNCTION

FUNCTION GLOBAL DSComm_Interface::UnsubscribeEventjournalUpdates

  DSComm.UnsubscribeEventjournalUpdates();

END_FUNCTION

FUNCTION GLOBAL DSComm_Interface::SubscribeUserEvents
	VAR_INPUT
		MajorID 	: UINT;
		MinorID 	: UINT;
	END_VAR
	VAR_OUTPUT
		ErrorNo 	: DINT;
	END_VAR

  ErrorNo := DSComm.SubscribeUserEvents(MajorID, MinorID, this);

END_FUNCTION

FUNCTION GLOBAL DSComm_Interface::UnsubscribeUserEvents
	VAR_INPUT
		MajorID 	: UINT;
		MinorID 	: UINT;
	END_VAR
	VAR_OUTPUT
		ErrorNo 	: DINT;
	END_VAR

  ErrorNo := DSComm.UnsubscribeUserEvents(MajorID, MinorID, this);

END_FUNCTION

FUNCTION GLOBAL DSComm_Interface::SetParameter
	VAR_INPUT
		ParaNo 	: DSComm::_DS_Parameter;
		Value 	: DINT;
		Mode 	: DINT;
	END_VAR
	VAR_OUTPUT
		Retcode 	: DINT;
	END_VAR

  Retcode := DSComm.SetParameter(ParaNo, Value, Mode);

END_FUNCTION

FUNCTION GLOBAL DSComm_Interface::GetParameter
	VAR_INPUT
		ParaNo 	: DSComm::_DS_Parameter;
		pValue 	: ^DINT;
		Mode 	: DINT;
	END_VAR
	VAR_OUTPUT
		Retcode 	: DINT;
	END_VAR

  Retcode := DSComm.GetParameter(ParaNo, pValue, Mode);

END_FUNCTION

FUNCTION GLOBAL DSComm_Interface::StartTCPComm

  DSComm.StartTCPComm();

END_FUNCTION

#pragma warning(disable: 73)
FUNCTION VIRTUAL GLOBAL DSComm_Interface::UserEventReceive
	VAR_INPUT
		MajorID 	: UINT;
		MinorID 	: UINT;
		MessageID 	: DINT;
		ErrorNo 	: DINT;
		pData 	: pVoid;
		Length 	: UDINT;
	END_VAR
#pragma warning(default: 73)

END_FUNCTION

FUNCTION VIRTUAL GLOBAL DSComm_Interface::Background
	VAR_INPUT
		EAX 	: UDINT;
	END_VAR
	VAR_OUTPUT
		state (EAX) 	: UDINT;
	END_VAR

	state := READY;

END_FUNCTION

#pragma warning(disable: 73)
FUNCTION VIRTUAL GLOBAL DSComm_Interface::AddLocalClientResp
	VAR_INPUT
		MessageID 	: DINT;
		ErrorNo 	: DINT;
		pAddLocalClientRsp 	: ^DSComm::_DS_AddLocalClientResp;
	END_VAR
#pragma warning(default: 73)

END_FUNCTION

#pragma warning(disable: 73)
FUNCTION VIRTUAL GLOBAL DSComm_Interface::AddLocalClientRangeResp
	VAR_INPUT
		MessageID 	: DINT;
		ErrorNo 	: DINT;
		pAddLocalClientRangeRsp 	: ^DSComm::_DS_AddLocalClientRangeResp;
	END_VAR
#pragma warning(default: 73)

END_FUNCTION

#pragma warning(disable: 73)
FUNCTION VIRTUAL GLOBAL DSComm_Interface::RemoveThisLocalClientResp
	VAR_INPUT
		MessageID 	: DINT;
		ErrorNo 	: DINT;
		pRemoveThisLocalClientRsp 	: ^DSComm::_DS_RemoveThisLocalClientResp;
	END_VAR
#pragma warning(default: 73)

END_FUNCTION

#pragma warning(disable: 73)
FUNCTION VIRTUAL GLOBAL DSComm_Interface::RemoveLocalClientResp
	VAR_INPUT
		MessageID 	: DINT;
		ErrorNo 	: DINT;
		pRemoveLocalClientRsp 	: ^DSComm::_DS_RemoveLocalClientResp;
	END_VAR
#pragma warning(default: 73)

END_FUNCTION

#pragma warning(disable: 73)
FUNCTION VIRTUAL GLOBAL DSComm_Interface::RemoveLocalClientRangeResp
	VAR_INPUT
		MessageID 	: DINT;
		ErrorNo 	: DINT;
		pRemoveLocalClientRangeRsp 	: ^DSComm::_DS_RemoveLocalClientRangeResp;
	END_VAR
#pragma warning(default: 73)

END_FUNCTION

#pragma warning(disable: 73)
FUNCTION VIRTUAL GLOBAL DSComm_Interface::ClearLocalClientListResp
	VAR_INPUT
		MessageID 	: DINT;
		ErrorNo 	: DINT;
		pClearLocalClientListRsp 	: ^DSComm::_DS_ClearLocalClientListResp;
	END_VAR
#pragma warning(default: 73)

END_FUNCTION

#pragma warning(disable: 73)
FUNCTION VIRTUAL GLOBAL DSComm_Interface::GetCurrentIDResp
	VAR_INPUT
		MessageID 	: DINT;
		ErrorNo 	: DINT;
		pGetCurrentIDRsp 	: ^DSComm::_DS_GetCurrentIDResp;
	END_VAR
#pragma warning(default: 73)

END_FUNCTION

#pragma warning(disable: 73)
FUNCTION VIRTUAL GLOBAL DSComm_Interface::GetLocalClientListResp
	VAR_INPUT
		MessageID 	: DINT;
		ErrorNo 	: DINT;
		num 	: UDINT;
		pGetLocalClientListRsp 	: ^DSComm::_DS_GetLocalClientListResp;
	END_VAR
#pragma warning(default: 73)

END_FUNCTION

#pragma warning(disable: 73)
FUNCTION VIRTUAL GLOBAL DSComm_Interface::GetLocalClientListDetailsResp
	VAR_INPUT
		MessageID 	: DINT;
		ErrorNo 	: DINT;
		num 	: UDINT;
		pGetLocalClientListDetailsRsp 	: ^DSComm::_DS_GetLocalClientDetailsResp;
	END_VAR
#pragma warning(default: 73)

END_FUNCTION

#pragma warning(disable: 73)
FUNCTION VIRTUAL GLOBAL DSComm_Interface::GetLocalClientByIDResp
	VAR_INPUT
		MessageID 	: DINT;
		ErrorNo 	: DINT;
		pGetLocalClientByIDRsp 	: ^DSComm::_DS_GetLocalClientDetailsResp;
	END_VAR
#pragma warning(default: 73)

END_FUNCTION

FUNCTION GLOBAL DSComm_Interface::GetProjectInfo
	VAR_OUTPUT
		MessageID 	: DINT;
	END_VAR

  MessageID := DSComm.GetProjectInfo(pThis:=this);
END_FUNCTION

FUNCTION GLOBAL DSComm_Interface::AddLocalClient
	VAR_INPUT
		pLocalClient 	: ^DSComm::_DS_AddLocalClientCmd;
	END_VAR
	VAR_OUTPUT
		MessageID 	: DINT;
	END_VAR

  MessageID := DSComm.AddLocalClient(pThis:=this, pLocalClient);
END_FUNCTION

FUNCTION GLOBAL DSComm_Interface::AddLocalClientRange
	VAR_INPUT
		pLocalClientRange 	: ^DSComm::_DS_AddLocalClientRangeCmd;
	END_VAR
	VAR_OUTPUT
		MessageID 	: DINT;
	END_VAR

  MessageID := DSComm.AddLocalClientRange(pThis:=this, pLocalClientRange);
END_FUNCTION

FUNCTION GLOBAL DSComm_Interface::GetCurrentID
	VAR_OUTPUT
		MessageID 	: DINT;
	END_VAR

  MessageID := DSComm.GetCurrentID(pThis:=this);
END_FUNCTION

FUNCTION GLOBAL DSComm_Interface::RemoveThisLocalClient
	VAR_OUTPUT
		MessageID 	: DINT;
	END_VAR

  MessageID := DSComm.RemoveThisLocalClient(pThis:=this);
END_FUNCTION

FUNCTION GLOBAL DSComm_Interface::RemoveLocalClient
	VAR_INPUT
		pLocalClient 	: ^DSComm::_DS_RemoveLocalClientCmd;
	END_VAR
	VAR_OUTPUT
		MessageID 	: DINT;
	END_VAR

  MessageID := DSComm.RemoveLocalClient(pThis:=this, pLocalClient);
END_FUNCTION

FUNCTION GLOBAL DSComm_Interface::RemoveLocalClientRange
	VAR_INPUT
		pLocalClientRange 	: ^DSComm::_DS_RemoveLocalClientRangeCmd;
	END_VAR
	VAR_OUTPUT
		MessageID 	: DINT;
	END_VAR

  MessageID := DSComm.RemoveLocalClientRange(pThis:=this, pLocalClientRange);
END_FUNCTION

FUNCTION GLOBAL DSComm_Interface::ClearLocalClientList
	VAR_OUTPUT
		MessageID 	: DINT;
	END_VAR

  MessageID := DSComm.ClearLocalClientList(pThis:=this);
END_FUNCTION

FUNCTION GLOBAL DSComm_Interface::GetLocalClientList
	VAR_OUTPUT
		MessageID 	: DINT;
	END_VAR

  MessageID := DSComm.GetLocalClientList(pThis:=this);
END_FUNCTION

FUNCTION GLOBAL DSComm_Interface::GetLocalClientListDetails
	VAR_OUTPUT
		MessageID 	: DINT;
	END_VAR

  MessageID := DSComm.GetLocalClientListDetails(pThis:=this);
END_FUNCTION

FUNCTION GLOBAL DSComm_Interface::GetLocalClientByID
	VAR_INPUT
		pLocalClient 	: ^DSComm::_DS_GetLocalClientByIDCmd;
	END_VAR
	VAR_OUTPUT
		MessageID 	: DINT;
	END_VAR

  MessageID := DSComm.GetLocalClientByID(pThis:=this, pLocalClient);
END_FUNCTION

FUNCTION GLOBAL DSComm_Interface::SubscribeAlarmListUpdate
	VAR_OUTPUT
		MessageID 	: DINT;
	END_VAR

  MessageID := DSComm.SubscribeAlarmListUpdate(pThis:=this);
END_FUNCTION

FUNCTION GLOBAL DSComm_Interface::UnsubscribeAlarmListUpdate
	VAR_OUTPUT
		MessageID 	: DINT;
	END_VAR

  MessageID := DSComm.UnsubscribeAlarmListUpdate(pThis:=this);
END_FUNCTION

#pragma warning(disable: 73)
FUNCTION VIRTUAL GLOBAL DSComm_Interface::SubscribeAlarmListUpdateResp
	VAR_INPUT
		MessageID 	: DINT;
		ErrorNo 	: DINT;
		pAlarmListUpdateAddRsp 	: ^DSComm::_DS_AlarmListUpdateAddResp;
	END_VAR
#pragma warning(default: 73)

END_FUNCTION

#pragma warning(disable: 73)
FUNCTION VIRTUAL GLOBAL DSComm_Interface::UnsubscribeAlarmListUpdateResp
	VAR_INPUT
		MessageID 	: DINT;
		ErrorNo 	: DINT;
		pAlarmListUpdateSubRsp 	: ^DSComm::_DS_AlarmListUpdateSubResp;
	END_VAR
#pragma warning(default: 73)

END_FUNCTION

#pragma warning(disable: 73)
FUNCTION VIRTUAL GLOBAL DSComm_Interface::AlarmListUpdatePush
	VAR_INPUT
		ErrorNo 	: DINT;
		num 	: UDINT;
		pAlarmListUpd 	: ^DSComm::_DS_AlarmListUpdate;
	END_VAR
#pragma warning(default: 73)

END_FUNCTION

FUNCTION GLOBAL DSComm_Interface::SubscribeHotAlarmUpdate
	VAR_INPUT
		pHotAlarm 	: ^DSComm::_DS_HotAlarmAddCmd;
	END_VAR
	VAR_OUTPUT
		MessageID 	: DINT;
	END_VAR

  MessageID := DSComm.SubscribeHotAlarmUpdate(pThis:=this, pHotAlarm);
END_FUNCTION

FUNCTION GLOBAL DSComm_Interface::UnsubscribeHotAlarmUpdate
	VAR_INPUT
		pHotAlarm 	: ^DSComm::_DS_HotAlarmSubCmd;
	END_VAR
	VAR_OUTPUT
		MessageID 	: DINT;
	END_VAR

  MessageID := DSComm.UnsubscribeHotAlarmUpdate(pThis:=this, pHotAlarm);
END_FUNCTION

#pragma warning(disable: 73)
FUNCTION VIRTUAL GLOBAL DSComm_Interface::SubscribeHotAlarmUpdateResp
	VAR_INPUT
		MessageID 	: DINT;
		ErrorNo 	: DINT;
		pHotAlarmUpdateAddRsp 	: ^DSComm::_DS_HotAlarmAddResp;
	END_VAR
#pragma warning(default: 73)

END_FUNCTION

#pragma warning(disable: 73)
FUNCTION VIRTUAL GLOBAL DSComm_Interface::UnsubscribeHotAlarmUpdateResp
	VAR_INPUT
		MessageID 	: DINT;
		ErrorNo 	: DINT;
		pHotAlarmUpdateSubRsp 	: ^DSComm::_DS_HotAlarmSubResp;
	END_VAR
#pragma warning(default: 73)

END_FUNCTION

#pragma warning(disable: 73)
FUNCTION VIRTUAL GLOBAL DSComm_Interface::HotAlarmUpdatePush
	VAR_INPUT
		ErrorNo 	: DINT;
		num 	: UDINT;
		pHotAlarmUpd 	: ^DSComm::_DS_HotAlarmUpdate;
	END_VAR
#pragma warning(default: 73)

END_FUNCTION

FUNCTION GLOBAL DSComm_Interface::AlarmDelete
	VAR_INPUT
		num 	: UDINT;
		toDelState 	: USINT;
		pAlarmID 	: ^UDINT;
	END_VAR
	VAR_OUTPUT
		MessageID 	: DINT;
	END_VAR

  MessageID := DSComm.AlarmDelete(pThis:=this, num, toDelState, pAlarmID);
END_FUNCTION

FUNCTION GLOBAL DSComm_Interface::AlarmDeleteAll
	VAR_INPUT
		toDelState 	: USINT;
	END_VAR
	VAR_OUTPUT
		MessageID 	: DINT;
	END_VAR

  MessageID := DSComm.AlarmDeleteAll(pThis:=this, toDelState);
END_FUNCTION

#pragma warning(disable: 73)
FUNCTION VIRTUAL GLOBAL DSComm_Interface::AlarmDeleteResp
	VAR_INPUT
		MessageID 	: DINT;
		ErrorNo 	: DINT;
		num 	: UDINT;
		pAlarmDeleteRsp 	: ^DSComm::_DS_AlarmDeleteResp;
	END_VAR
#pragma warning(default: 73)

END_FUNCTION

#pragma warning(disable: 73)
FUNCTION VIRTUAL GLOBAL DSComm_Interface::AlarmDeleteAllResp
	VAR_INPUT
		MessageID 	: DINT;
		ErrorNo 	: DINT;
		pAlarmDeleteAllRsp 	: ^DSComm::_DS_AlarmDeleteAllResp;
	END_VAR
#pragma warning(default: 73)

END_FUNCTION

#pragma warning(disable: 73)
FUNCTION VIRTUAL GLOBAL DSComm_Interface::AlarmDeleteUpdatePush
	VAR_INPUT
		ErrorNo 	: DINT;
		num 	: UDINT;
		pAlarmDeleteUpd 	: ^DSComm::_DS_AlarmDeleteUpdate;
	END_VAR
#pragma warning(default: 73)

END_FUNCTION

FUNCTION GLOBAL DSComm_Interface::StrLenUtf8
	VAR_INPUT
		Str_Utf8 	: ^CHAR;
	END_VAR
	VAR_OUTPUT
		retcode 	: UDINT;
	END_VAR

  retcode := DSComm.StrLenUtf8(Str_Utf8);

END_FUNCTION

#pragma warning(disable: 73)
FUNCTION VIRTUAL GLOBAL DSComm_Interface::SubscribeStateResp
	VAR_INPUT
		MessageID 	: DINT;
		ErrorNo 	: DINT;
		pSubscribeStateRsp 	: ^DSComm::_DS_SubscribeStateResp;
	END_VAR
#pragma warning(default: 73)

END_FUNCTION

#pragma warning(disable: 73)
FUNCTION VIRTUAL GLOBAL DSComm_Interface::UnsubscribeStateResp
	VAR_INPUT
		MessageID 	: DINT;
		ErrorNo 	: DINT;
		pUnsubscribeStateRsp 	: ^DSComm::_DS_UnsubscribeStateResp;
	END_VAR
#pragma warning(default: 73)

END_FUNCTION

#pragma warning(disable: 73)
FUNCTION VIRTUAL GLOBAL DSComm_Interface::Get_StateResp
	VAR_INPUT
		MessageID 	: DINT;
		ErrorNo 	: DINT;
		pGetStateRsp 	: ^DSComm::_DS_GetStateResp;
	END_VAR
#pragma warning(default: 73)

END_FUNCTION

#pragma warning(disable: 73)
FUNCTION VIRTUAL GLOBAL DSComm_Interface::UpdateStatePush
	VAR_INPUT
		pUpdateState 	: ^DSComm::_DS_GetStateResp;
	END_VAR
#pragma warning(default: 73)

END_FUNCTION

FUNCTION GLOBAL DSComm_Interface::SubscribeState
	VAR_INPUT
		pCmdData 	: ^DSComm::_DS_SubscribeStateCmd;
	END_VAR
	VAR_OUTPUT
		MessageID 	: DINT;
	END_VAR

  MessageID := DSComm.SubscribeState(pThis:=this, pCmdData);
END_FUNCTION

FUNCTION GLOBAL DSComm_Interface::UnsubscribeState
	VAR_INPUT
		pCmdData 	: ^DSComm::_DS_UnsubscribeStateCmd;
	END_VAR
	VAR_OUTPUT
		MessageID 	: DINT;
	END_VAR

  MessageID := DSComm.UnsubscribeState(pThis:=this, pCmdData);
END_FUNCTION

FUNCTION GLOBAL DSComm_Interface::Get_State
	VAR_INPUT
		pCmdData 	: ^DSComm::_DS_GetStateCmd;
	END_VAR
	VAR_OUTPUT
		MessageID 	: DINT;
	END_VAR

  MessageID := DSComm.Get_State(pThis:=this, pCmdData);
END_FUNCTION
